(* CODESYS project load_stand.project

Project tree, tasks and I/O mapping:
  Device : Owen SPK2xx 03.CS.WEB, Owen, order no. 023, version 3.5.4.20
    application Application
      libraries: Standard, * (System); Util, 3.5.1.0 (System); CmpSysExec, 1.0.0.2 (Owen)
      task MainTask (cyclic, interval t#100ms, priority 2) calls Main_PRG
      task VISU_TASK (cyclic, interval 100 ms, priority 30) calls VisuElems.Visu_Prg
      task AlarmManagerTask (cyclic, interval 50 ms, priority 31) calls AlarmManager.Alarm_Prg
      task bus_task (cyclic, interval t#100ms, priority 1, watchdog t#1000ms x 1) calls nothing
      program PLC_PRG [ST]
      function block Two_words_to_Real [ST]
      visualisation mpx_1_params
      image pool ImagePool
      program Main_PRG [ST]
      visualisation mpx_2_params
      visualisation main
      program InterviewState [ST]
      visualisation mu_a3
      text list TextList
    Modbus_COM : Modbus COM, 3S - Smart Software Solutions GmbH, version 3.4.0.0
        settings: DataBits = 8; StopBits = 1; ComPort = 4
      Modbus_Master_COM_Port : Modbus Master, COM Port, 3S - Smart Software Solutions GmbH, version 3.5.5.0
          settings: Transmission = 'RTU'; ResponseTimeout = 1000; TimeBetweenFrames = 10; Auto-restart communication = TRUE
        MU_A3 : Modbus Slave, COM Port, 3S - Smart Software Solutions GmbH, version 3.5.4.0
            settings: SlaveAddress = 3; ResponseTimeout = 1000; UseExtendedFunctionCodes = TRUE; Channel 0.Function Code = 16; Channel 0.Read Offset = 0; Channel 0.Read Length = 0; Channel 0.Write Offset = 16#0061; Channel 0.Write Length = 2; Channel 0.Cycle Time = 500
            output Application.Main_PRG.mu_a3_states_2 : WORD  // Channel 0.Channel 0
            output Application.Main_PRG.mu_a3_states_1 : WORD  // Channel 0.Channel 0
            unmapped channels: Channel 0
        MU_A2 : Modbus Slave, COM Port, 3S - Smart Software Solutions GmbH, version 3.5.4.0
            settings: SlaveAddress = 2; ResponseTimeout = 1000; UseExtendedFunctionCodes = TRUE; Channel 0.Function Code = 16; Channel 0.Read Offset = 0; Channel 0.Read Length = 0; Channel 0.Write Offset = 16#0061; Channel 0.Write Length = 2; Channel 0.Cycle Time = 500
            output Application.Main_PRG.mu_a2_states_2 : WORD  // Channel 0.Channel 0
            output Application.Main_PRG.mu_a2_states_1 : WORD  // Channel 0.Channel 0
            unmapped channels: Channel 0
  text list GlobalTextList
  5ce3da45-db07-42e7-a21c-a00fff4ed8f6|C:\workspace\UGP\Images\schrpa.png
  5ce3da45-db07-42e7-a21c-a00fff4ed8f6|D:\scheme_3.png
  5ce3da45-db07-42e7-a21c-a00fff4ed8f6|C:\workspace\UGP\Images\bg_800.png
  5ce3da45-db07-42e7-a21c-a00fff4ed8f6|D:\scheme.png
  5ce3da45-db07-42e7-a21c-a00fff4ed8f6|D:\on.png
  5ce3da45-db07-42e7-a21c-a00fff4ed8f6|D:\off.png
  5ce3da45-db07-42e7-a21c-a00fff4ed8f6|D:\off.jpg
  5ce3da45-db07-42e7-a21c-a00fff4ed8f6|D:\on.jpg
  5ce3da45-db07-42e7-a21c-a00fff4ed8f6|D:\on_ind.jpg
  5ce3da45-db07-42e7-a21c-a00fff4ed8f6|D:\off_ind.jpg
  5ce3da45-db07-42e7-a21c-a00fff4ed8f6|D:\entel.png
  5ce3da45-db07-42e7-a21c-a00fff4ed8f6|D:\zit.png
  5ce3da45-db07-42e7-a21c-a00fff4ed8f6|D:\entel.jpg
  5ce3da45-db07-42e7-a21c-a00fff4ed8f6|D:\zit.jpg
  5ce3da45-db07-42e7-a21c-a00fff4ed8f6|D:\vvod_off.png
  5ce3da45-db07-42e7-a21c-a00fff4ed8f6|D:\vvod_on.png
  5ce3da45-db07-42e7-a21c-a00fff4ed8f6|C:\workspace\UGP\Images\bg.png
  5ce3da45-db07-42e7-a21c-a00fff4ed8f6|C:\workspace\UGP\Images\ups_800.png
  5ce3da45-db07-42e7-a21c-a00fff4ed8f6|C:\workspace\UGP\Images\ups\ups_800.png
  5ce3da45-db07-42e7-a21c-a00fff4ed8f6|C:\workspace\UGP\Images\ups\bypass_line1_off.png
  5ce3da45-db07-42e7-a21c-a00fff4ed8f6|C:\workspace\UGP\Images\ups\bypass_arrow_off.png
  5ce3da45-db07-42e7-a21c-a00fff4ed8f6|C:\workspace\UGP\Images\ups\arrow_off.png
  5ce3da45-db07-42e7-a21c-a00fff4ed8f6|C:\workspace\UGP\Images\ups\battery_arrow_off.png
  5ce3da45-db07-42e7-a21c-a00fff4ed8f6|C:\workspace\UGP\Images\ups\battery_line_off.png
  5ce3da45-db07-42e7-a21c-a00fff4ed8f6|C:\workspace\UGP\Images\ups\battery_arrow_on.png
  5ce3da45-db07-42e7-a21c-a00fff4ed8f6|C:\workspace\UGP\Images\ups\bypass_line_on.png
  5ce3da45-db07-42e7-a21c-a00fff4ed8f6|C:\workspace\UGP\Images\ups\bypass_arrow_on.png
  5ce3da45-db07-42e7-a21c-a00fff4ed8f6|C:\workspace\UGP\Images\ups\arrow_on.png
  5ce3da45-db07-42e7-a21c-a00fff4ed8f6|C:\workspace\UGP\Images\ups\battery_line_on.png
  5ce3da45-db07-42e7-a21c-a00fff4ed8f6|C:\workspace\UGP\Images\main_bg.png
  5ce3da45-db07-42e7-a21c-a00fff4ed8f6|C:\workspace\UGP\Images\shasn.png
  5ce3da45-db07-42e7-a21c-a00fff4ed8f6|C:\workspace\UGP\Images\shasn_1.png
  5ce3da45-db07-42e7-a21c-a00fff4ed8f6|C:\workspace\UGP\Images\ips_state_bg.png
  5ce3da45-db07-42e7-a21c-a00fff4ed8f6|C:\workspace\UGP\Images\mpx_state_bg.png
  5ce3da45-db07-42e7-a21c-a00fff4ed8f6|C:\workspace\UGP\Images\shasn_800.png
*)

// Device/Application/Main_PRG
PROGRAM Main_PRG
VAR
	mu_a2_states_1        :WORD:=0;
	mu_a2_states_1_bit    :BIT_AS_WORD;
	mu_a2_states_1_bits   :ARRAY[0..15] of BOOL;
	
	mu_a2_states_2        :WORD:=0;
	mu_a2_states_2_bit    :BIT_AS_WORD;
	mu_a2_states_2_bits   :ARRAY[0..15] OF BOOL;
	
	mu_a3_states_1        :WORD:=0;
	mu_a3_states_1_bit    :BIT_AS_WORD;
	mu_a3_states_1_bits   :ARRAY[0..15] OF BOOL;
	
	mu_a3_states_2        :WORD:=0;
	mu_a3_states_2_bit    :BIT_AS_WORD;
	mu_a3_states_2_bits   :ARRAY[0..15] OF BOOL;
	
	list :WORD;
END_VAR

mu_a2_states_1_bit(B00 := mu_a2_states_1_bits[0], 
                   B01 := mu_a2_states_1_bits[1],
				   B02 := mu_a2_states_1_bits[2],
				   B03 := mu_a2_states_1_bits[3],
				   B04 := mu_a2_states_1_bits[4],
				   B05 := mu_a2_states_1_bits[5],
				   B06 := mu_a2_states_1_bits[6],
				   B07 := mu_a2_states_1_bits[7],
				   B08 := mu_a2_states_1_bits[8],
				   B09 := mu_a2_states_1_bits[9],
				   B10 := mu_a2_states_1_bits[10],
				   B11 := mu_a2_states_1_bits[11],
				   B12 := mu_a2_states_1_bits[12],
				   B13 := mu_a2_states_1_bits[13],
				   B14 := mu_a2_states_1_bits[14],
				   B15 := mu_a2_states_1_bits[15]
                  );				  
mu_a2_states_1 := mu_a2_states_1_bit.W;

mu_a2_states_2_bit(B00 := mu_a2_states_2_bits[0], 
                   B01 := mu_a2_states_2_bits[1],
				   B02 := mu_a2_states_2_bits[2],
				   B03 := mu_a2_states_2_bits[3],
				   B04 := mu_a2_states_2_bits[4],
				   B05 := mu_a2_states_2_bits[5],
				   B06 := mu_a2_states_2_bits[6],
				   B07 := mu_a2_states_2_bits[7],
				   B08 := mu_a2_states_2_bits[8],
				   B09 := mu_a2_states_2_bits[9],
				   B10 := mu_a2_states_2_bits[10],
				   B11 := mu_a2_states_2_bits[11],
				   B12 := mu_a2_states_2_bits[12],
				   B13 := mu_a2_states_2_bits[13],
				   B14 := mu_a2_states_2_bits[14],
				   B15 := mu_a2_states_2_bits[15]
                  );				  
mu_a2_states_2 := mu_a2_states_2_bit.W;

mu_a3_states_1_bit(B00 := mu_a3_states_1_bits[0], 
                   B01 := mu_a3_states_1_bits[1],
				   B02 := mu_a3_states_1_bits[2],
				   B03 := mu_a3_states_1_bits[3],
				   B04 := mu_a3_states_1_bits[4],
				   B05 := mu_a3_states_1_bits[5],
				   B06 := mu_a3_states_1_bits[6],
				   B07 := mu_a3_states_1_bits[7],
				   B08 := mu_a3_states_1_bits[8],
				   B09 := mu_a3_states_1_bits[9],
				   B10 := mu_a3_states_1_bits[10],
				   B11 := mu_a3_states_1_bits[11],
				   B12 := mu_a3_states_1_bits[12],
				   B13 := mu_a3_states_1_bits[13],
				   B14 := mu_a3_states_1_bits[14],
				   B15 := mu_a3_states_1_bits[15]
                  );				  
mu_a3_states_1 := mu_a3_states_1_bit.W;

mu_a3_states_2_bit(B00 := mu_a3_states_2_bits[0], 
                   B01 := mu_a3_states_2_bits[1],
				   B02 := mu_a3_states_2_bits[2],
				   B03 := mu_a3_states_2_bits[3],
				   B04 := mu_a3_states_2_bits[4],
				   B05 := mu_a3_states_2_bits[5],
				   B06 := mu_a3_states_2_bits[6],
				   B07 := mu_a3_states_2_bits[7],
				   B08 := mu_a3_states_2_bits[8],
				   B09 := mu_a3_states_2_bits[9],
				   B10 := mu_a3_states_2_bits[10],
				   B11 := mu_a3_states_2_bits[11],
				   B12 := mu_a3_states_2_bits[12],
				   B13 := mu_a3_states_2_bits[13],
				   B14 := mu_a3_states_2_bits[14],
				   B15 := mu_a3_states_2_bits[15]
                  );				  
mu_a3_states_2 := mu_a3_states_2_bit.W;

END_PROGRAM

// Device/Application/PLC_PRG
PROGRAM PLC_PRG
VAR
	




	var_test :BOOL:=false;
	alm_1: BOOL;
	alm_2: BOOL;
	war_1: BOOL;
	war_2: BOOL;
	//Переменные для отработки аварийных ситуаций
	accident_sectional_machine :BOOL := FALSE; //авария секционного автомата
	accident_input_1		   :BOOL := FALSE; //авария ввода №1
	accident_input_2		   :BOOL := FALSE; //авария ввода №2
	accident_no_voltage_in_1   :BOOL := FALSE; //отсутствие напряжения на вводе №1
	accident_no_voltage_in_2   :BOOL := FALSE; //отсутствие напряжения на вводе №2
	manual_mode				   :BOOL := FALSE;
	accident_no_voltage_sec    :BOOL := FALSE; //отсутствие напряжения на секции
	
	var_off : BOOL := FALSE;
	var_on : BOOL := TRUE;
	
	//Визуализация
	var_true :BOOL := TRUE;
	ack		 :BOOL;
	history  :BOOL;
	
	//Переменные для работы с MPX_1
	mpx1_in_v_1 	 		   		:WORD; //1-е Напрядение входа
	mpx1_in_v_2 	 		   		:WORD; //2-e Напряжение входа
	mpx1_in_v_3 	 		   		:WORD; //3-е Напряжение входа
	mpx1_in_freq 	 		   		:WORD; //Частота на входе
	mpx1_in_freq_real		   		:REAL; //Частота на входе (x0.1)
	mpx1_bypass_v_1  		   		:WORD; //1-е Напряжение байпаса
	mpx1_bypass_v_2  		   		:WORD; //2-е Напряжение байпаса
	mpx1_bypass_v_3  		   		:WORD; //3-е Напряжение байпаса
	mpx1_bypass_freq 		   		:WORD; //Частота байпаса
	mpx1_bypass_freq_real      		:REAL; //Частота байпаса
	mpx1_output_v_1  		   		:WORD; //1-е Напряжение выхода
	mpx1_output_v_2  		   		:WORD; //2-е Напряжение выхода
	mpx1_output_v_3  		   		:WORD; //3-е Напряжение выхода
	mpx1_output_i_1  		   		:WORD; //1-й Ток выхода
	mpx1_output_i_2  		   		:WORD; //2-й Ток выхода
	mpx1_output_i_3  		   		:WORD; //3-й Ток выхода
	mpx1_output_i_1_real       		:REAL; //1-й Ток выхода (x0.1)
	mpx1_output_i_2_real       		:REAL; //2-й Ток выхода (x0.1)
	mpx1_output_i_3_real       		:REAL; //3-й Ток выхода (x0.1)
	mpx1_output_active_power_1 		:WORD; //Активная мощность 1-й фазы
	mpx1_output_active_power_2 		:WORD; //Активная мощность 2-й фазы
	mpx1_output_active_power_3 		:WORD; //Активная мощность 3-й фазы
	mpx1_output_active_power_1_real :REAL; //Активная мощность 1-й фазы (x0.1)
	mpx1_output_active_power_2_real :REAL; //Активная мощность 2-й фазы (x0.1)
	mpx1_output_active_power_3_real :REAL; //Активная мощность 3-й фазы (x0.1)
	mpx1_output_freq 	       		:WORD; //Частота выхода
	mpx1_output_freq_real 	        :REAL; //Частота выхода (x0.1)
	mpx1_load_ph_1    	       		:WORD; //Загрузска 1-й фазы (%)
	mpx1_load_ph_2    		   		:WORD; //Загрузска 3-й фазы (%)
	mpx1_load_ph_3    	       		:WORD; //Загрузска 2-й фазы (%)
	mpx1_battery_voltage 	   		:WORD; //Напряжение батареи
	mpx1_battery_voltage_real  		:REAL; //Напряжение батареи (x0.1)
	mpx1_battery_current 	   		:WORD; //Ток батареи
	mpx1_battery_current_real  		:REAL; //Ток батареи (x0.1)
	mpx1_battery_capacity 	   		:WORD; //Остаточная емкость батареи (%)
	mpx1_battery_time 		   		:WORD; //Остаточное время автономии (минуты)
	mpx1_temp 				   		:WORD; //Температура
	mpx1_state_reg_1 	       		:WORD; //1-й Регистр состояния
	mpx1_state_1_as_bit 	   		:WORD_AS_BIT;
	mpx1_state_reg_2 		   		:WORD; //2-й Регистр состояния
	mpx1_state_2_as_bit 	   		:WORD_AS_BIT;
	mpx1_bypass_line_state 	   		:STRING; 
	mpx1_bypass_arrow_state    		:STRING;
	mpx1_battery_arrow_state 		:STRING; //состояние батареи
	mpx1_battery_line_state 		:STRING; //состояние батареи
	mpx1_input_state 		   		:STRING; //состояние входа
	mpx1_output_state 		   		:STRING; //состояние выхода
	mpx1_alarm                      :BOOL;
	mpx_test_battery_command        :WORD:=20;
	mpx_test_battery_start          :BOOL;
		
	//Переменные для работы с MPX_2
	mpx2_in_v_1 	 		   		:WORD; //1-е Напрядение входа
	mpx2_in_v_2 	 		   		:WORD; //2-e Напряжение входа
	mpx2_in_v_3 	 		   		:WORD; //3-е Напряжение входа
	mpx2_in_freq 	 		   		:WORD; //Частота на входе
	mpx2_in_freq_real		   		:REAL; //Частота на входе (x0.1)
	mpx2_bypass_v_1  		   		:WORD; //1-е Напряжение байпаса
	mpx2_bypass_v_2  		   		:WORD; //2-е Напряжение байпаса
	mpx2_bypass_v_3  		   		:WORD; //3-е Напряжение байпаса
	mpx2_bypass_freq 		   		:WORD; //Частота байпаса
	mpx2_bypass_freq_real      		:REAL; //Частота байпаса
	mpx2_output_v_1  		   		:WORD; //1-е Напряжение выхода
	mpx2_output_v_2  		   		:WORD; //2-е Напряжение выхода
	mpx2_output_v_3  		   		:WORD; //3-е Напряжение выхода
	mpx2_output_i_1  		   		:WORD; //1-й Ток выхода
	mpx2_output_i_2  		   		:WORD; //2-й Ток выхода
	mpx2_output_i_3  		   		:WORD; //3-й Ток выхода
	mpx2_output_i_1_real       		:REAL; //1-й Ток выхода (x0.1)
	mpx2_output_i_2_real       		:REAL; //2-й Ток выхода (x0.1)
	mpx2_output_i_3_real       		:REAL; //3-й Ток выхода (x0.1)
	mpx2_output_active_power_1 		:WORD; //Активная мощность 1-й фазы
	mpx2_output_active_power_2 		:WORD; //Активная мощность 2-й фазы
	mpx2_output_active_power_3 		:WORD; //Активная мощность 3-й фазы
	mpx2_output_active_power_1_real :REAL; //Активная мощность 1-й фазы (x0.1)
	mpx2_output_active_power_2_real :REAL; //Активная мощность 2-й фазы (x0.1)
	mpx2_output_active_power_3_real :REAL; //Активная мощность 3-й фазы (x0.1)
	mpx2_output_freq 	       		:WORD; //Частота выхода
	mpx2_output_freq_real 	        :REAL; //Частота выхода (x0.1)
	mpx2_load_ph_1    	       		:WORD; //Загрузска 1-й фазы (%)
	mpx2_load_ph_2    		   		:WORD; //Загрузска 3-й фазы (%)
	mpx2_load_ph_3    	       		:WORD; //Загрузска 2-й фазы (%)
	mpx2_battery_voltage 	   		:WORD; //Напряжение батареи
	mpx2_battery_voltage_real  		:REAL; //Напряжение батареи (x0.1)
	mpx2_battery_current 	   		:WORD; //Ток батареи
	mpx2_battery_current_real  		:REAL; //Ток батареи (x0.1)
	mpx2_battery_capacity 	   		:WORD; //Остаточная емкость батареи (%)
	mpx2_battery_time 		   		:WORD; //Остаточное время автономии (минуты)
	mpx2_temp 				   		:WORD; //Температура
	mpx2_state_reg_1 	       		:WORD; //1-й Регистр состояния
	mpx2_state_1_as_bit 	   		:WORD_AS_BIT;
	mpx2_state_reg_2 		   		:WORD; //2-й Регистр состояния
	mpx2_state_2_as_bit 	   		:WORD_AS_BIT;
	mpx2_bypass_line_state 	   		:STRING; 
	mpx2_bypass_arrow_state    		:STRING;
	mpx2_battery_arrow_state 		:STRING; //состояние батареи
	mpx2_battery_line_state 		:STRING; //состояние батареи
	mpx2_input_state 		   		:STRING; //состояние входа
	mpx2_output_state 		   		:STRING; //состояние выхода
	mpx2_alarm                      :BOOL;
	
	//Переменные для работы с климатом
	climate_temp_out        :WORD;
	climat_temp_out_minus   :BOOL; //Регистр отрицательности температуры
	climate_temp_out_real   :REAL;
	climate_temp_in         :WORD;
	climat_temp_in_minus    :BOOL; //Регистр отрицательности температуры
	climate_temp_in_real    :REAL;
	climate_state_reg       :WORD;
	climate_state_as_bit    :WORD_AS_BIT;
	climate_zaslonka_state  :BOOL;
	climate_vent_state      :BOOL;
	climate_condition_state :BOOL;
	climate_heat_state      :BOOL;
	climate_auto_state      :BOOL;
	climate_temp_excess     :BOOL; //авария. внутренняя температура > 25
	
	//Переменные для работы с IPS_1
	ips1_in_v_1           :WORD; //1-е Напряжение входа
	ips1_in_v_1_real      :REAL;
	ips1_in_v_2           :WORD; //2-е Напряжение входа
	ips1_in_v_2_real      :REAL;
	ips1_in_v_3           :WORD; //3-е Напряжение входа
	ips1_in_v_3_real      :REAL;
	ips1_bypass_v         :WORD; //Напряжение байпаса
	ips1_bypass_v_real    :REAL;
	ips1_out_v            :WORD; //Выходное напряжение
	ips1_out_v_real       :REAL;
	ips1_out_freq         :WORD; //Выходная частота
	ips1_out_freq_real    :REAL;
	ips1_out_load         :WORD; //Выходная загрузка
	ips1_out_load_real    :REAL;
	ips1_battery_v        :WORD; //Напряжение батареи
	ips1_battery_v_real   :REAL;
	ips1_battery_capacity :WORD; //Емкость батареи
	ips1_battery_i        :WORD;
	ips1_battery_i_real   :REAL; //Ток батареи
	
	//Переменные для работы с IPS_2
	ips2_in_v_1           :WORD; //1-е Напряжение входа
	ips2_in_v_1_real      :REAL;
	ips2_in_v_2           :WORD; //2-е Напряжение входа
	ips2_in_v_2_real      :REAL;
	ips2_in_v_3           :WORD; //3-е Напряжение входа
	ips2_in_v_3_real      :REAL;
	ips2_bypass_v         :WORD; //Напряжение байпаса
	ips2_bypass_v_real    :REAL;
	ips2_out_v            :WORD; //Выходное напряжение
	ips2_out_v_real       :REAL;
	ips2_out_freq         :WORD; //Выходная частота
	ips2_out_freq_real    :REAL;
	ips2_out_load         :WORD; //Выходная загрузка
	ips2_out_load_real    :REAL;
	ips2_battery_v        :WORD; //Напряжение батареи
	ips2_battery_v_real   :REAL;
	ips2_battery_capacity :WORD; //Емкость батареи
	ips2_battery_i        :WORD;
	ips2_battery_i_real   :REAL; //Ток батареи
	
	//Переменные для работы с первым МВ110-16 (адрес = 1)
	mv110_reg	                   :WORD; //Регистр состояния входов МВ110-16
	mv110_reg_as_bit 	           :WORD_AS_BIT; 
	mv110_in_0_alarm_shos 		   :BOOL; //Нарушение ШОС
	mv110_in_1_fire 			   :BOOL; //Пожар
	mv110_in_2_alarm_ops 		   :BOOL; //Авария ОПС
	mv110_in_3_shasn_main_input    :BOOL; //ШАСН напряжение на основном вводе
	mv110_in_4_shasn_reserve_input :BOOL; //ШАСН напряжение на резервном вводе
	mv110_in_5_shasn_right         :BOOL; //ШАСН напряжение на правой шине
	mv110_in_6_shasn_left          :BOOL; //ШАСН напряжение на левой шине
	mv110_in_7_heating 	           :BOOL; //Обогрев включен
	mv110_in_8_shasn_main 	           :BOOL; //ШАСН основной ввод
	mv110_in_9_shasn_reserve 	           :BOOL; //ШАСН резервный ввод
	mv110_in_10_schrpa_main_input  :BOOL; //ЩРПА напряжение на основном вводе
	mv110_in_11_schrpa_reserve_input  :BOOL; //ЩРПА напряжение на резервном вводе
	mv110_in_12_manual_bypass_1_1   :BOOL; //ЩРПА Ручной байпас 1.1
	mv110_in_12_manual_bypass_1_2  :BOOL; //ЩРПА Ручной байпас 1.2
	
	//Переменные ЩРПА
	schrpa_avr_left_on   :BOOL;
	schrpa_avr_right_on  :BOOL;
	
END_VAR

//Конвертация параметров mpx_1
mpx1_in_freq_real     := mpx1_in_freq * 0.1;
mpx1_bypass_freq_real := mpx1_bypass_freq * 0.1;
mpx1_output_i_1_real  := mpx1_output_i_1 * 0.1;
mpx1_output_i_2_real  := mpx1_output_i_2 * 0.1;
mpx1_output_i_3_real  := mpx1_output_i_3 * 0.1;
mpx1_output_active_power_1_real := mpx1_output_active_power_1 * 0.1;
mpx1_output_active_power_2_real := mpx1_output_active_power_2 * 0.1;
mpx1_output_active_power_3_real := mpx1_output_active_power_3 * 0.1;
mpx1_output_freq_real := mpx1_output_freq * 0.1;
mpx1_battery_voltage_real := mpx1_battery_voltage * 0.1;
mpx1_battery_current_real := mpx1_battery_current * 0.1;

//Логика состояний mpx_1
mpx1_state_1_as_bit(W := mpx1_state_reg_1);
mpx1_state_2_as_bit(W := mpx1_state_reg_2);
IF (mpx1_state_1_as_bit.B11 = FALSE) THEN
	mpx1_bypass_line_state := 'bypass_line1_off';
	mpx1_bypass_arrow_state := 'bypass_arrow_off';
	ELSE
		mpx1_bypass_line_state := 'bypass_line_on';
		mpx1_bypass_arrow_state := 'bypass_arrow_on';	
END_IF
IF (mpx1_state_1_as_bit.B15 = FALSE) THEN
	mpx1_output_state := 'arrow_off';
	ELSE
		mpx1_output_state := 'arrow_on';	
END_IF
IF (mpx1_state_2_as_bit.B12 = FALSE) THEN
	mpx1_input_state := 'arrow_off';
	ELSE
		mpx1_input_state := 'arrow_on';	
END_IF
IF (mpx1_state_1_as_bit.B13 = FALSE) THEN
	mpx1_battery_line_state := 'battery_line_off';
	mpx1_battery_arrow_state := 'battery_arrow_off';
	ELSE
		mpx1_battery_line_state := 'battery_line_on';
		mpx1_battery_arrow_state := 'battery_arrow_on';	
END_IF
IF ( (mpx1_state_2_as_bit.B13 = TRUE) OR (mpx1_state_2_as_bit.B14 = TRUE) OR (mpx1_state_2_as_bit.B15 = TRUE) ) THEN
	mpx1_alarm := TRUE;
	ELSE
		mpx1_alarm := FALSE;
END_IF

//Конвертация параметров mpx_2
mpx2_in_freq_real               := mpx2_in_freq * 0.1;
mpx2_bypass_freq_real           := mpx2_bypass_freq * 0.1;
mpx2_output_i_1_real            := mpx2_output_i_1 * 0.1;
mpx2_output_i_2_real            := mpx2_output_i_2 * 0.1;
mpx2_output_i_3_real            := mpx2_output_i_3 * 0.1;
mpx2_output_active_power_1_real := mpx2_output_active_power_1 * 0.1;
mpx2_output_active_power_2_real := mpx2_output_active_power_2 * 0.1;
mpx2_output_active_power_3_real := mpx2_output_active_power_3 * 0.1;
mpx2_output_freq_real           := mpx2_output_freq * 0.1;
mpx2_battery_voltage_real       := mpx2_battery_voltage * 0.1;
mpx2_battery_current_real       := mpx2_battery_current * 0.1;

//Логика состояний mpx_2
mpx2_state_1_as_bit(W := mpx2_state_reg_1);
mpx2_state_2_as_bit(W := mpx2_state_reg_2);
IF (mpx2_state_1_as_bit.B11 = FALSE) THEN
	mpx2_bypass_line_state := 'bypass_line1_off';
	mpx2_bypass_arrow_state := 'bypass_arrow_off';
	ELSE
		mpx2_bypass_line_state := 'bypass_line_on';
		mpx2_bypass_arrow_state := 'bypass_arrow_on';	
END_IF
IF (mpx2_state_1_as_bit.B15 = FALSE) THEN
	mpx2_output_state := 'arrow_off';
	ELSE
		mpx2_output_state := 'arrow_on';	
END_IF
IF (mpx2_state_2_as_bit.B12 = FALSE) THEN
	mpx2_input_state := 'arrow_off';
	ELSE
		mpx2_input_state := 'arrow_on';	
END_IF
IF (mpx2_state_1_as_bit.B13 = FALSE) THEN
	mpx2_battery_line_state := 'battery_line_off';
	mpx2_battery_arrow_state := 'battery_arrow_off';
	ELSE
		mpx2_battery_line_state := 'battery_line_on';
		mpx2_battery_arrow_state := 'battery_arrow_on';	
END_IF
IF ( (mpx2_state_2_as_bit.B13 = TRUE) OR (mpx2_state_2_as_bit.B14 = TRUE) OR (mpx2_state_2_as_bit.B15 = TRUE) ) THEN
	mpx2_alarm := TRUE;
	ELSE
		mpx2_alarm := FALSE;
END_IF

//Работа с климатом
climate_state_as_bit(W  := climate_state_reg);
climate_zaslonka_state  := climate_state_as_bit.B03;
climate_vent_state      := climate_state_as_bit.B00;
climate_condition_state := climate_state_as_bit.B01;
climate_heat_state      := climate_state_as_bit.B02;
climate_auto_state      := climate_state_as_bit.B04;
climat_temp_out_minus   := climate_state_as_bit.B07;
climat_temp_in_minus    := climate_state_as_bit.B06;
climate_temp_out_real   := climate_temp_out * 0.1;
climate_temp_in_real    := climate_temp_in * 0.1;
IF (climat_temp_out_minus = TRUE) THEN
	climate_temp_out_real := climate_temp_out_real * (-1);
END_IF
IF (climat_temp_in_minus = TRUE) THEN
	climate_temp_in_real := climate_temp_in_real * (-1);
END_IF
IF (climate_temp_in_real > 25) THEN
	climate_temp_excess := TRUE;
	ELSE
		climate_temp_excess := FALSE;
END_IF

//Конвертация ips_1
ips1_in_v_1_real    := ips1_in_v_1 * 0.1;
ips1_in_v_2_real    := ips1_in_v_2 * 0.1;
ips1_in_v_3_real    := ips1_in_v_3 * 0.1;
ips1_bypass_v_real  := ips1_bypass_v * 0.1;
ips1_out_v_real     := ips1_out_v * 0.1;
ips1_out_freq_real  := ips1_out_freq * 0.1;
ips1_battery_v_real := ips1_battery_v * 0.1;
ips1_battery_i_real := ips1_battery_i * 0.1;
ips1_out_load_real  := ips1_out_load * 0.1;

//Конвертация ips_2
ips2_in_v_1_real    := ips2_in_v_1 * 0.1;
ips2_in_v_2_real    := ips2_in_v_2 * 0.1;
ips2_in_v_3_real    := ips2_in_v_3 * 0.1;
ips2_bypass_v_real  := ips2_bypass_v * 0.1;
ips2_out_v_real     := ips2_out_v * 0.1;
ips2_out_freq_real  := ips2_out_freq * 0.1;
ips2_battery_v_real := ips2_battery_v * 0.1;
ips2_battery_i_real := ips2_battery_i * 0.1;
ips2_out_load_real  := ips2_out_load * 0.1;

//Логика МВ110-16
mv110_reg_as_bit(W := mv110_reg);
mv110_in_0_alarm_shos          := mv110_reg_as_bit.B00;
mv110_in_1_fire                := mv110_reg_as_bit.B01;
mv110_in_2_alarm_ops           := mv110_reg_as_bit.B02;
mv110_in_3_shasn_main_input    := mv110_reg_as_bit.B03;
mv110_in_4_shasn_reserve_input := mv110_reg_as_bit.B04;
mv110_in_5_shasn_right         := mv110_reg_as_bit.B05;
mv110_in_6_shasn_left          := mv110_reg_as_bit.B06;
mv110_in_7_heating             := mv110_reg_as_bit.B07;
mv110_in_8_shasn_main             := mv110_reg_as_bit.B08;
mv110_in_9_shasn_reserve             := mv110_reg_as_bit.B09;
mv110_in_10_schrpa_main_input  := mv110_reg_as_bit.B10;
mv110_in_11_schrpa_reserve_input  := mv110_reg_as_bit.B11;
mv110_in_12_manual_bypass_1_1  := mv110_reg_as_bit.B12;
mv110_in_12_manual_bypass_1_2  := mv110_reg_as_bit.B13;

//Логика ЩРПА
IF (mv110_in_10_schrpa_main_input = TRUE) THEN
	schrpa_avr_left_on := TRUE;
	schrpa_avr_right_on := FALSE;
END_IF
IF ( (mv110_in_10_schrpa_main_input = FALSE) AND (mv110_in_11_schrpa_reserve_input = TRUE) ) THEN
	schrpa_avr_left_on := FALSE;
	schrpa_avr_right_on := TRUE;
END_IF
IF ( (mv110_in_10_schrpa_main_input = FALSE) AND (mv110_in_11_schrpa_reserve_input = FALSE) ) THEN
	schrpa_avr_left_on := FALSE;
	schrpa_avr_right_on := FALSE;
END_IF

//Пример конвертации
//module_v1_u1_convertion(Inpit_1:=module_v1_u1_reg1 , Inpit_2:=module_v1_u1_reg2 , output=>module_v1_u1 ); //V1 Ua

END_PROGRAM

// Device/Application/Two_words_to_Real
FUNCTION_BLOCK Two_words_to_Real
VAR_INPUT
	Inpit_1:WORD;
	Inpit_2:WORD;
END_VAR
VAR_OUTPUT
	output:real;
END_VAR
VAR
	P:POINTER TO ARRAY [0..3] OF BYTE; 
	pi1:POINTER TO ARRAY [0..1] OF BYTE; 
	pi2:POINTER TO ARRAY [0..1] OF BYTE; 
END_VAR

pi1:=ADR(Inpit_1);
pi2:=ADR(Inpit_2);



P:=ADR(output);
P^[0]:=pi2^[0];
P^[1]:=pi2^[1];
P^[2]:=pi1^[0];
P^[3]:=pi1^[1];

END_FUNCTION_BLOCK

// Device/Application/InterviewState
PROGRAM InterviewState
VAR
(*	MV110_err :BOOL;
	MPX1_err :BOOL;
	MPX2_err :BOOL;
	IPS1_err :BOOL;
	IPS2_err :BOOL;*)
END_VAR

(*IF (MV110.xError = TRUE) THEN
	MV110_err := TRUE;
	ELSE
		MV110_err := FALSE;
END_IF

IF (MPX_1.xError = TRUE) THEN
	MPX1_err := TRUE;
	ELSE
		MPX1_err := FALSE;
END_IF

IF (MPX_2.xError = TRUE) THEN
	MPX2_err := TRUE;
	ELSE
		MPX2_err := FALSE;
END_IF

IF (IPS_1.xError = TRUE) THEN
	IPS1_err := TRUE;
	ELSE
		IPS1_err := FALSE;
END_IF

IF (IPS_2.xError = TRUE) THEN
	IPS2_err := TRUE;
	ELSE
		IPS2_err := FALSE;
END_IF
*)

END_PROGRAM

// Device/Application/mpx_1_params
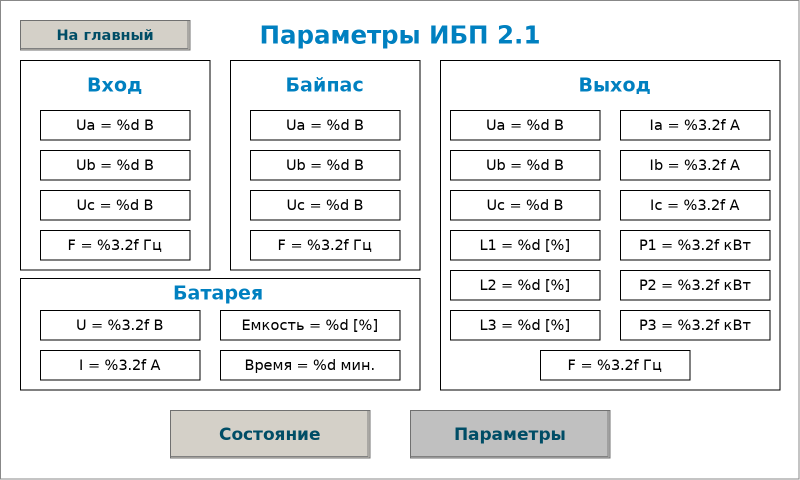
VISUALIZATION mpx_1_params  // 800x480, background image ImagePool.bg_800
    Rectangle (186,20 428x30), "Параметры ИБП 2.1"
    Button (170,410 200x48), "Состояние"
        OnMouseClick:  Assign=mpx_1_state, Type=Assignment
    Button (410,410 200x48), "Параметры", pressed state: PLC_PRG.var_true
    Button (20,20 170x30), "На главный"
        OnMouseClick:  Assign=main, Type=Assignment
    Rectangle (20,60 190x210)
    Rectangle (440,60 340x330)
    Rectangle (30,70 170x30), "Вход"
    Rectangle (40,110 150x30), "Ua = %d В", text variable: PLC_PRG.mpx1_in_v_1
    Rectangle (40,150 150x30), "Ub = %d В", text variable: PLC_PRG.mpx1_in_v_2
    Rectangle (40,190 150x30), "Uc = %d В", text variable: PLC_PRG.mpx1_in_v_3
    Rectangle (40,230 150x30), "F = %3.2f Гц", text variable: PLC_PRG.mpx1_in_freq_real
    Rectangle (230,60 190x210)
    Rectangle (240,70 170x30), "Байпас"
    Rectangle (250,110 150x30), "Ua = %d В", text variable: PLC_PRG.mpx1_bypass_v_1
    Rectangle (250,150 150x30), "Ub = %d В", text variable: PLC_PRG.mpx1_bypass_v_2
    Rectangle (250,190 150x30), "Uc = %d В", text variable: PLC_PRG.mpx1_bypass_v_3
    Rectangle (250,230 150x30), "F = %3.2f Гц", text variable: PLC_PRG.mpx1_bypass_freq_real
    Rectangle (460,70 310x30), "Выход"
    Rectangle (450,110 150x30), "Ua = %d В", text variable: PLC_PRG.mpx1_output_v_1
    Rectangle (450,150 150x30), "Ub = %d В", text variable: PLC_PRG.mpx1_output_v_2
    Rectangle (450,190 150x30), "Uc = %d В", text variable: PLC_PRG.mpx1_output_v_3
    Rectangle (620,110 150x30), "Ia = %3.2f A", text variable: PLC_PRG.mpx1_output_i_1_real
    Rectangle (620,150 150x30), "Ib = %3.2f A", text variable: PLC_PRG.mpx1_output_i_2_real
    Rectangle (620,190 150x30), "Ic = %3.2f A", text variable: PLC_PRG.mpx1_output_i_3_real
    Rectangle (450,230 150x30), "L1 = %d [%]", text variable: PLC_PRG.mpx1_load_ph_1
    Rectangle (450,270 150x30), "L2 = %d [%]", text variable: PLC_PRG.mpx1_load_ph_2
    Rectangle (450,310 150x30), "L3 = %d [%]", text variable: PLC_PRG.mpx1_load_ph_3
    Rectangle (620,230 150x30), "P1 = %3.2f кВт", text variable: PLC_PRG.mpx1_output_active_power_1_real
    Rectangle (620,270 150x30), "P2 = %3.2f кВт", text variable: PLC_PRG.mpx1_output_active_power_2_real
    Rectangle (620,310 150x30), "P3 = %3.2f кВт", text variable: PLC_PRG.mpx1_output_active_power_3_real
    Rectangle (540,350 150x30), "F = %3.2f Гц", text variable: PLC_PRG.mpx1_output_freq_real
    Rectangle (20,278 400x112)
    Rectangle (30,284 376x18), "Батарея"
    Rectangle (40,310 160x30), "U = %3.2f В", text variable: PLC_PRG.mpx1_battery_voltage_real
    Rectangle (40,350 160x30), "I = %3.2f A", text variable: PLC_PRG.mpx1_battery_current_real
    Rectangle (220,310 180x30), "Емкость = %d [%]", text variable: PLC_PRG.mpx1_battery_capacity
    Rectangle (220,350 180x30), "Время = %d мин.", text variable: PLC_PRG.mpx1_battery_time
    hotkey  Id=481037385728, Key=KeyDown=True, KeyName=0
    hotkey  Id=481038434304, Key=KeyName=0
END_VISUALIZATION

// Device/Application/mpx_2_params
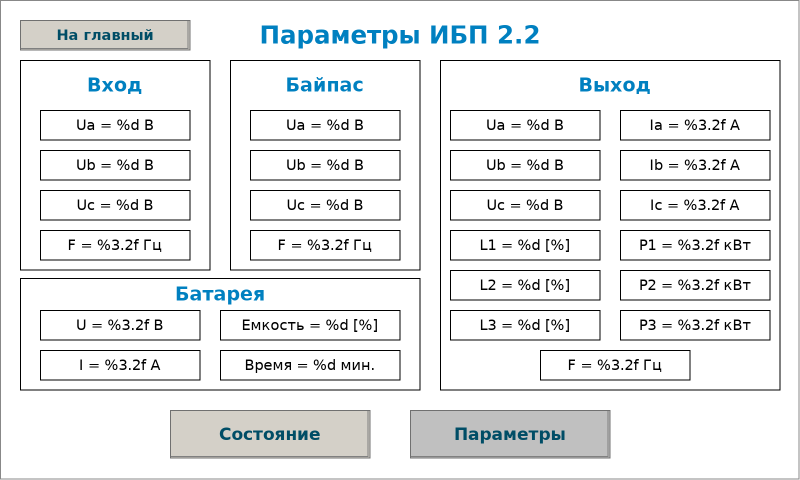
VISUALIZATION mpx_2_params  // 800x480, background image ImagePool.bg_800
    Rectangle (186,20 428x30), "Параметры ИБП 2.2"
    Button (170,410 200x48), "Состояние"
        OnMouseClick:  Assign=mpx_2_state, Type=Assignment
    Button (410,410 200x48), "Параметры", pressed state: PLC_PRG.var_true
    Button (20,20 170x30), "На главный"
        OnMouseClick:  Assign=main, Type=Assignment
    Rectangle (20,60 190x210)
    Rectangle (440,60 340x330)
    Rectangle (30,70 170x30), "Вход"
    Rectangle (40,110 150x30), "Ua = %d В", text variable: PLC_PRG.mpx2_in_v_1
    Rectangle (40,150 150x30), "Ub = %d В", text variable: PLC_PRG.mpx2_in_v_2
    Rectangle (40,190 150x30), "Uc = %d В", text variable: PLC_PRG.mpx2_in_v_3
    Rectangle (40,230 150x30), "F = %3.2f Гц", text variable: PLC_PRG.mpx2_in_freq_real
    Rectangle (230,60 190x210)
    Rectangle (240,70 170x30), "Байпас"
    Rectangle (250,110 150x30), "Ua = %d В", text variable: PLC_PRG.mpx2_bypass_v_1
    Rectangle (250,150 150x30), "Ub = %d В", text variable: PLC_PRG.mpx2_bypass_v_2
    Rectangle (250,190 150x30), "Uc = %d В", text variable: PLC_PRG.mpx2_bypass_v_3
    Rectangle (250,230 150x30), "F = %3.2f Гц", text variable: PLC_PRG.mpx2_bypass_freq_real
    Rectangle (460,70 310x30), "Выход"
    Rectangle (450,110 150x30), "Ua = %d В", text variable: PLC_PRG.mpx2_output_v_1
    Rectangle (450,150 150x30), "Ub = %d В", text variable: PLC_PRG.mpx2_output_v_2
    Rectangle (450,190 150x30), "Uc = %d В", text variable: PLC_PRG.mpx2_output_v_3
    Rectangle (620,110 150x30), "Ia = %3.2f A", text variable: PLC_PRG.mpx2_output_i_1_real
    Rectangle (620,150 150x30), "Ib = %3.2f A", text variable: PLC_PRG.mpx2_output_i_2_real
    Rectangle (620,190 150x30), "Ic = %3.2f A", text variable: PLC_PRG.mpx2_output_i_3_real
    Rectangle (450,230 150x30), "L1 = %d [%]", text variable: PLC_PRG.mpx2_load_ph_1
    Rectangle (450,270 150x30), "L2 = %d [%]", text variable: PLC_PRG.mpx2_load_ph_2
    Rectangle (450,310 150x30), "L3 = %d [%]", text variable: PLC_PRG.mpx2_load_ph_3
    Rectangle (620,230 150x30), "P1 = %3.2f кВт", text variable: PLC_PRG.mpx2_output_active_power_1_real
    Rectangle (620,270 150x30), "P2 = %3.2f кВт", text variable: PLC_PRG.mpx2_output_active_power_2_real
    Rectangle (620,310 150x30), "P3 = %3.2f кВт", text variable: PLC_PRG.mpx2_output_active_power_3_real
    Rectangle (540,350 150x30), "F = %3.2f Гц", text variable: PLC_PRG.mpx2_output_freq_real
    Rectangle (20,278 400x112)
    Rectangle (30,282 380x24), "Батарея"
    Rectangle (40,310 160x30), "U = %3.2f В", text variable: PLC_PRG.mpx2_battery_voltage_real
    Rectangle (40,350 160x30), "I = %3.2f A", text variable: PLC_PRG.mpx2_battery_current_real
    Rectangle (220,310 180x30), "Емкость = %d [%]", text variable: PLC_PRG.mpx2_battery_capacity
    Rectangle (220,350 180x30), "Время = %d мин.", text variable: PLC_PRG.mpx2_battery_time
    hotkey  Id=481037385728, Key=KeyDown=True, KeyName=0
    hotkey  Id=481038434304, Key=KeyName=0
END_VISUALIZATION

// Device/Application/main
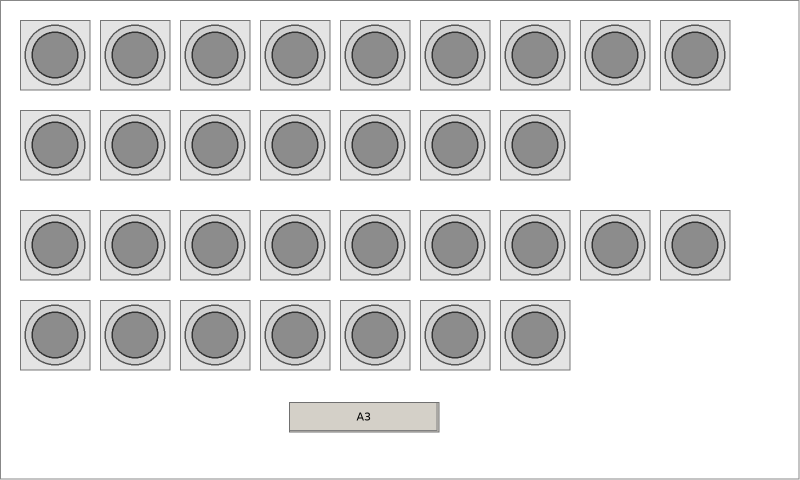
VISUALIZATION main  // 800x480, background image ImagePool.bg_800
    PushSwitchLed (20,20 70x70), variable: Main_PRG.mu_a2_states_1_bits[0], behaviour: TOGGLE, style: Switch-PushSwitchLed-Gray
    PushSwitchLed (100,20 70x70), variable: Main_PRG.mu_a2_states_1_bits[1], behaviour: TOGGLE, style: Switch-PushSwitchLed-Gray
    PushSwitchLed (180,20 70x70), variable: Main_PRG.mu_a2_states_1_bits[2], behaviour: TOGGLE, style: Switch-PushSwitchLed-Gray
    PushSwitchLed (260,20 70x70), variable: Main_PRG.mu_a2_states_1_bits[3], behaviour: TOGGLE, style: Switch-PushSwitchLed-Gray
    PushSwitchLed (340,20 70x70), variable: Main_PRG.mu_a2_states_1_bits[4], behaviour: TOGGLE, style: Switch-PushSwitchLed-Gray
    PushSwitchLed (420,20 70x70), variable: Main_PRG.mu_a2_states_1_bits[5], behaviour: TOGGLE, style: Switch-PushSwitchLed-Gray
    PushSwitchLed (500,20 70x70), variable: Main_PRG.mu_a2_states_1_bits[6], behaviour: TOGGLE, style: Switch-PushSwitchLed-Gray
    PushSwitchLed (580,20 70x70), variable: Main_PRG.mu_a2_states_1_bits[7], behaviour: TOGGLE, style: Switch-PushSwitchLed-Gray
    PushSwitchLed (660,20 70x70), variable: Main_PRG.mu_a2_states_1_bits[8], behaviour: TOGGLE, style: Switch-PushSwitchLed-Gray
    PushSwitchLed (20,110 70x70), variable: Main_PRG.mu_a2_states_1_bits[9], behaviour: TOGGLE, style: Switch-PushSwitchLed-Gray
    PushSwitchLed (100,110 70x70), variable: Main_PRG.mu_a2_states_1_bits[10], behaviour: TOGGLE, style: Switch-PushSwitchLed-Gray
    PushSwitchLed (180,110 70x70), variable: Main_PRG.mu_a2_states_1_bits[11], behaviour: TOGGLE, style: Switch-PushSwitchLed-Gray
    PushSwitchLed (260,110 70x70), variable: Main_PRG.mu_a2_states_1_bits[12], behaviour: TOGGLE, style: Switch-PushSwitchLed-Gray
    PushSwitchLed (340,110 70x70), variable: Main_PRG.mu_a2_states_1_bits[13], behaviour: TOGGLE, style: Switch-PushSwitchLed-Gray
    PushSwitchLed (420,110 70x70), variable: Main_PRG.mu_a2_states_1_bits[14], behaviour: TOGGLE, style: Switch-PushSwitchLed-Gray
    PushSwitchLed (500,110 70x70), variable: Main_PRG.mu_a2_states_1_bits[15], behaviour: TOGGLE, style: Switch-PushSwitchLed-Gray
    PushSwitchLed (20,210 70x70), variable: Main_PRG.mu_a2_states_2_bits[0], behaviour: TOGGLE, style: Switch-PushSwitchLed-Gray
    PushSwitchLed (100,210 70x70), variable: Main_PRG.mu_a2_states_2_bits[1], behaviour: TOGGLE, style: Switch-PushSwitchLed-Gray
    PushSwitchLed (180,210 70x70), variable: Main_PRG.mu_a2_states_2_bits[2], behaviour: TOGGLE, style: Switch-PushSwitchLed-Gray
    PushSwitchLed (260,210 70x70), variable: Main_PRG.mu_a2_states_2_bits[3], behaviour: TOGGLE, style: Switch-PushSwitchLed-Gray
    PushSwitchLed (340,210 70x70), variable: Main_PRG.mu_a2_states_2_bits[4], behaviour: TOGGLE, style: Switch-PushSwitchLed-Gray
    PushSwitchLed (420,210 70x70), variable: Main_PRG.mu_a2_states_2_bits[5], behaviour: TOGGLE, style: Switch-PushSwitchLed-Gray
    PushSwitchLed (500,210 70x70), variable: Main_PRG.mu_a2_states_2_bits[6], behaviour: TOGGLE, style: Switch-PushSwitchLed-Gray
    PushSwitchLed (580,210 70x70), variable: Main_PRG.mu_a2_states_2_bits[7], behaviour: TOGGLE, style: Switch-PushSwitchLed-Gray
    PushSwitchLed (660,210 70x70), variable: Main_PRG.mu_a2_states_2_bits[8], behaviour: TOGGLE, style: Switch-PushSwitchLed-Gray
    PushSwitchLed (20,300 70x70), variable: Main_PRG.mu_a2_states_2_bits[9], behaviour: TOGGLE, style: Switch-PushSwitchLed-Gray
    PushSwitchLed (100,300 70x70), variable: Main_PRG.mu_a2_states_2_bits[10], behaviour: TOGGLE, style: Switch-PushSwitchLed-Gray
    PushSwitchLed (180,300 70x70), variable: Main_PRG.mu_a2_states_2_bits[11], behaviour: TOGGLE, style: Switch-PushSwitchLed-Gray
    PushSwitchLed (260,300 70x70), variable: Main_PRG.mu_a2_states_2_bits[12], behaviour: TOGGLE, style: Switch-PushSwitchLed-Gray
    PushSwitchLed (340,300 70x70), variable: Main_PRG.mu_a2_states_2_bits[13], behaviour: TOGGLE, style: Switch-PushSwitchLed-Gray
    PushSwitchLed (420,300 70x70), variable: Main_PRG.mu_a2_states_2_bits[14], behaviour: TOGGLE, style: Switch-PushSwitchLed-Gray
    PushSwitchLed (500,300 70x70), variable: Main_PRG.mu_a2_states_2_bits[15], behaviour: TOGGLE, style: Switch-PushSwitchLed-Gray
    Button (289,402 150x30), "A3"
        OnMouseClick:  Assign=mu_a3, Type=Assignment
END_VISUALIZATION

// Device/Application/mu_a3
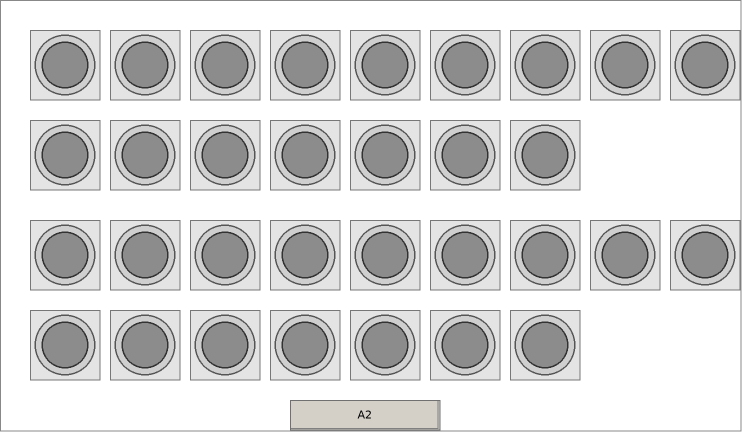
VISUALIZATION mu_a3  // 742x432
    PushSwitchLed (30,30 70x70), variable: Main_PRG.mu_a3_states_1_bits[0], behaviour: TOGGLE, style: Switch-PushSwitchLed-Gray
    PushSwitchLed (110,30 70x70), variable: Main_PRG.mu_a3_states_1_bits[1], behaviour: TOGGLE, style: Switch-PushSwitchLed-Gray
    PushSwitchLed (190,30 70x70), variable: Main_PRG.mu_a3_states_1_bits[2], behaviour: TOGGLE, style: Switch-PushSwitchLed-Gray
    PushSwitchLed (270,30 70x70), variable: Main_PRG.mu_a3_states_1_bits[3], behaviour: TOGGLE, style: Switch-PushSwitchLed-Gray
    PushSwitchLed (350,30 70x70), variable: Main_PRG.mu_a3_states_1_bits[4], behaviour: TOGGLE, style: Switch-PushSwitchLed-Gray
    PushSwitchLed (430,30 70x70), variable: Main_PRG.mu_a3_states_1_bits[5], behaviour: TOGGLE, style: Switch-PushSwitchLed-Gray
    PushSwitchLed (510,30 70x70), variable: Main_PRG.mu_a3_states_1_bits[6], behaviour: TOGGLE, style: Switch-PushSwitchLed-Gray
    PushSwitchLed (590,30 70x70), variable: Main_PRG.mu_a3_states_1_bits[7], behaviour: TOGGLE, style: Switch-PushSwitchLed-Gray
    PushSwitchLed (670,30 70x70), variable: Main_PRG.mu_a3_states_1_bits[8], behaviour: TOGGLE, style: Switch-PushSwitchLed-Gray
    PushSwitchLed (30,120 70x70), variable: Main_PRG.mu_a3_states_1_bits[9], behaviour: TOGGLE, style: Switch-PushSwitchLed-Gray
    PushSwitchLed (110,120 70x70), variable: Main_PRG.mu_a3_states_1_bits[10], behaviour: TOGGLE, style: Switch-PushSwitchLed-Gray
    PushSwitchLed (190,120 70x70), variable: Main_PRG.mu_a3_states_1_bits[11], behaviour: TOGGLE, style: Switch-PushSwitchLed-Gray
    PushSwitchLed (270,120 70x70), variable: Main_PRG.mu_a3_states_1_bits[12], behaviour: TOGGLE, style: Switch-PushSwitchLed-Gray
    PushSwitchLed (350,120 70x70), variable: Main_PRG.mu_a3_states_1_bits[13], behaviour: TOGGLE, style: Switch-PushSwitchLed-Gray
    PushSwitchLed (430,120 70x70), variable: Main_PRG.mu_a3_states_1_bits[14], behaviour: TOGGLE, style: Switch-PushSwitchLed-Gray
    PushSwitchLed (510,120 70x70), variable: Main_PRG.mu_a3_states_1_bits[15], behaviour: TOGGLE, style: Switch-PushSwitchLed-Gray
    PushSwitchLed (30,220 70x70), variable: Main_PRG.mu_a3_states_2_bits[0], behaviour: TOGGLE, style: Switch-PushSwitchLed-Gray
    PushSwitchLed (110,220 70x70), variable: Main_PRG.mu_a3_states_2_bits[1], behaviour: TOGGLE, style: Switch-PushSwitchLed-Gray
    PushSwitchLed (190,220 70x70), variable: Main_PRG.mu_a3_states_2_bits[2], behaviour: TOGGLE, style: Switch-PushSwitchLed-Gray
    PushSwitchLed (270,220 70x70), variable: Main_PRG.mu_a3_states_2_bits[3], behaviour: TOGGLE, style: Switch-PushSwitchLed-Gray
    PushSwitchLed (350,220 70x70), variable: Main_PRG.mu_a3_states_2_bits[4], behaviour: TOGGLE, style: Switch-PushSwitchLed-Gray
    PushSwitchLed (430,220 70x70), variable: Main_PRG.mu_a3_states_2_bits[5], behaviour: TOGGLE, style: Switch-PushSwitchLed-Gray
    PushSwitchLed (510,220 70x70), variable: Main_PRG.mu_a3_states_2_bits[6], behaviour: TOGGLE, style: Switch-PushSwitchLed-Gray
    PushSwitchLed (590,220 70x70), variable: Main_PRG.mu_a3_states_2_bits[7], behaviour: TOGGLE, style: Switch-PushSwitchLed-Gray
    PushSwitchLed (670,220 70x70), variable: Main_PRG.mu_a3_states_2_bits[8], behaviour: TOGGLE, style: Switch-PushSwitchLed-Gray
    PushSwitchLed (30,310 70x70), variable: Main_PRG.mu_a3_states_2_bits[9], behaviour: TOGGLE, style: Switch-PushSwitchLed-Gray
    PushSwitchLed (110,310 70x70), variable: Main_PRG.mu_a3_states_2_bits[10], behaviour: TOGGLE, style: Switch-PushSwitchLed-Gray
    PushSwitchLed (190,310 70x70), variable: Main_PRG.mu_a3_states_2_bits[11], behaviour: TOGGLE, style: Switch-PushSwitchLed-Gray
    PushSwitchLed (270,310 70x70), variable: Main_PRG.mu_a3_states_2_bits[12], behaviour: TOGGLE, style: Switch-PushSwitchLed-Gray
    PushSwitchLed (350,310 70x70), variable: Main_PRG.mu_a3_states_2_bits[13], behaviour: TOGGLE, style: Switch-PushSwitchLed-Gray
    PushSwitchLed (430,310 70x70), variable: Main_PRG.mu_a3_states_2_bits[14], behaviour: TOGGLE, style: Switch-PushSwitchLed-Gray
    PushSwitchLed (510,310 70x70), variable: Main_PRG.mu_a3_states_2_bits[15], behaviour: TOGGLE, style: Switch-PushSwitchLed-Gray
    Button (290,400 150x30), "A2"
        OnMouseClick:  Assign=main, Type=Assignment
END_VISUALIZATION

(* text list TextList (id | default)
  1 | 1
  2 | 2
  3 | 3
  4 | 4
  5 | 5
  6 | 6
  7 | 7
  8 | 8
  9 | 9
  10 | 10
   |  *)
